(* Schneider Machine Expert - Basic project modulus, file version 3.0.0.0 *)
(* ProjectInformations: Name=Nuovo progetto *)

HARDWARE
  Cpu 0: TM221CE40R
  EthernetConfiguration: NetworkName=M221, IpAllocationMode=FixedAddress, IpAddress=0.0.0.0, SubnetMask=0.0.0.0
  SerialLineConfiguration: Baud=Baud19200, Parity=ParityEven, DataBits=DataBits8, StopBits=StopBits1, PhysicalMedium=PhysicalMediumRs485, TransmissionMode=TransmissionModeModbusRtu, SlaveId=1, Addressing=SlaveAddressing
  MastTask: UsePeriodScanMode=false, PeriodScan=100
  FastTask: Period=255
  CpuBehavior: StartingMode=StartAsPreviousState, AutoSaveRamOnEeprom=true, WatchdogPeriod=250

SYMBOLS  (address, symbol, comment, settings)
  %MW2      REMAINDER
  %IW0.0    DIVIDEND  [Type=Type_0_10V, Scope=Scope_Normal, Minimum=0, Maximum=1000]
  %IW0.1    DIVISOR  [Type=Type_0_10V, Scope=Scope_Normal, Minimum=0, Maximum=1000]

POU Nuovo POU
  (* SectionNumber=1 *)

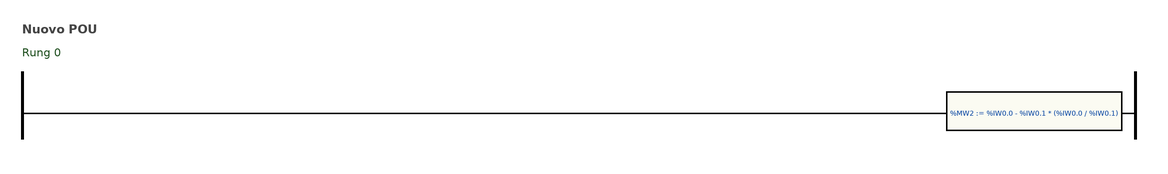

// Rung 0
  LD 1
  [ %MW2 := %IW0.0 - %IW0.1 * ( %IW0.0 / %IW0.1 ) ](* REMAINDER, DIVIDEND, DIVISOR, DIVIDEND, DIVISOR *)
  // as ST:
  //   REMAINDER := DIVIDEND - DIVISOR * ( DIVIDEND / DIVISOR );
